Universal Robots PolyScope program: SocketTCP_ex_nums.urp

Program interfaces_m3t2 (installation=default directory=/programs/usbdisk createdIn=5.11.1 lastSavedIn=5.13.1 robotSerialNumber=20205500771)
Calibrated DH parameters: a=[0.00017, -0.315777, -0.390584, 0.000089, 0.000022, 0]; d=[0.16289, -151.810109, 155.986099, -4.043122, 0.099816, 0.099706]; alpha=[1.572969, -0.001875, 0.009547, 1.571313, -1.570827, 0]; deltaTheta=[0, 0.733614, -0.631905, -0.101721, 0.000001, 0]
InitVariablesNode
BeforeStart
  'Interfaces Module 3 Task 2'
  'receive 2 values, add those values together, send the result back to the server'
  conn := False
  counter := 0
  progress := False
Robot Program (runOnlyOnce=true)
  Folder establish connection
    Loop While (checkContinuously=false) expression=conn≟ False
      conn := socket_open("192.168.0.12", 1701, "soc_name")
      Wait Sleep waitTime=2
      counter := counter+1
      progress := True
      Wait Sleep waitTime=5
      str := "ready"
      Script: socket_send_string(str, "soc_name")
      Script: socket_send_byte(13, "soc_name")
      Script: socket_send_byte(10, "soc_name")
  Wait Sleep waitTime=1
  Folder ask for the two values
    str := "what are the two numbers? format the numbers a and b as: (a, b)"
    Script: socket_send_string(str, "soc_name")
    Script: socket_send_byte(13, "soc_name")
    Script: socket_send_byte(10, "soc_name")
  Wait Sleep waitTime=1
  Folder read in the two numbers
    num_intake := [0,0,0]
    Loop While (checkContinuously=false) expression=num_intake[0]≟0
      num_intake := socket_read_ascii_float(2, "soc_name")
      Wait Sleep waitTime=0.1
    num_1 := num_intake[1]
    num_2 := num_intake[2]
    str := "numbers recieved "
    Script: socket_send_string(str, "soc_name")
    Script: socket_send_byte(13, "soc_name")
    Script: socket_send_byte(10, "soc_name")
  Wait Sleep waitTime=1
  Folder calculate resoponse and send
    total := to_str(num_1+num_2)
    Script: socket_send_string("the answer is: ", "soc_name")
    Script: socket_send_string(total, "soc_name")
    Script: socket_send_byte(13, "soc_name")
    Script: socket_send_byte(10, "soc_name")
  Wait Sleep waitTime=5
  Script: socket_close()
